(* PLC project shuttle, Dassault Systèmes ControlBuild 2024x *)
(* stored: creationDateTime 2023-10-03T11:13:56-01:00 *)

FUNCTION_BLOCK tri_chain.shuttle
  VAR_INPUT
    speedX : REAL := 0.0;
    speedY : REAL := 0.0;
  END_VAR
  VAR
    status_act_prod : DINT := 0;
    m11 : REAL := 1.0;
    m12 : REAL := 0.0;
    m13 : REAL := 0.0;
    m14 : REAL := 0.0;
    m21 : REAL := 0.0;
    m22 : REAL := 1.0;
    m23 : REAL := 0.0;
    m24 : REAL := 0.0;
    m31 : REAL := 0.0;
    m32 : REAL := 0.0;
    m33 : REAL := 1.0;
    m34 : REAL := 0.0;
    m41 : REAL := 0.0;
    m42 : REAL := 0.0;
    m43 : REAL := 0.0;
    m44 : REAL := 1.0;
    px : REAL := 0.0;
    py : REAL := 0.0;
    pz : REAL := 0.0;
    dx : REAL := 0.0;
    dy : REAL := 0.0;
    dz : REAL := 0.0;
    sProdX : REAL := 0.0;
    sProdY : REAL := 0.0;
  END_VAR
  VAR
    d_locking : BOOL := false;
    v_d_locking : BOOL := false;
  END_VAR


ACTION C_source_code:
/* ----------------------------------------------------------------	*/
/* Type : Model of Operative Behaviour					*/
/* Category :  Conveyor							*/
/* Author : Dassault Systemes						*/
/* Update date : June 2018							*/
/* ----------------------------------------------------------------	*/

/* -----------------------------------------------------------------	*/
/* px, py et pz are the lowest coordinates.				*/
/* dx, dy et dz are the actor's dimensions 				*/
/* sProdX is the speed given to the product for the X axis.		*/
/* sProdY s the speed given to the product for the Y axis.		*/
/* The linear speed is given in mm/s.					*/
/* -----------------------------------------------------------------	*/

/* -----------------------------------------------------------------	*/
/* The cyclic pitch  in function of the simulation cycle time		*/
/*		250 ms by default.						*/
/*	CLOCK_PERIOD returns the cycle time in 1000th. of ms		*/
/* -----------------------------------------------------------------	*/
if (!d_locking)
	{
	sProdX=speedX*(CLOCK_PERIOD/1000000);
	sProdY=speedY*(CLOCK_PERIOD/1000000);
	}
else 
	{
	sProdX=0;
	sProdY=0;
	}

px = px + sProdX;

moveTo(myself, px, py, pz);
END_ACTION
END_FUNCTION_BLOCK
